Yaskawa INFORM job: R1_W49-52-A5(180,0)KM-OK.JBI

/JOB
//NAME R1_W49-52-A5(180,0)KM-OK
///FOLDERNAME KRIS-SCIANA
//POS
///NPOS 116,116,0,8,0,0
///TOOL 0
///POSTYPE PULSE
///PULSE
C00000=236346,-93771,-119067,-15606,106110,52447
C00001=224522,-84676,-111717,21504,108396,-36823
C00002=223323,-76354,-80310,30853,97883,-38151
C00003=223323,-76354,-80296,30852,97876,-38153
C00004=224728,-76958,-80577,30799,97249,-37774
C00005=223323,-76354,-80296,30852,97876,-38153
C00006=223323,-76341,-79339,30801,97373,-38291
C00007=223323,-76354,-80296,30852,97876,-38153
C00008=212037,-83911,-83077,30593,100081,-41994
C00009=212037,-83786,-81846,30518,99482,-42157
C00010=212037,-83911,-83077,30593,100081,-41994
C00011=241412,-119790,-112905,4528,90278,-34927
C00012=241412,-120659,-108380,4524,87055,-35044
C00013=241412,-118950,-107832,4524,87594,-35023
C00014=241412,-120659,-108380,4524,87055,-35044
C00015=241361,-125463,-113452,4527,87710,-35038
C00016=194879,-88434,-95721,7341,99248,-50176
C00017=197359,-87135,-94304,7246,98826,-49360
C00018=197775,-85843,-93756,7239,99114,-49203
C00019=197359,-87135,-94304,7246,98826,-49360
C00020=197359,-86577,-97024,7299,100771,-49245
C00021=203638,-64502,-86768,7203,105226,-46867
C00022=203638,-66884,-80001,7025,99877,-47180
C00023=203638,-66998,-79410,7014,99457,-47204
C00024=203638,-66468,-81766,7061,101167,-47106
C00025=189796,-64404,-88301,-2122,101648,-53086
C00026=192138,-63897,-80248,-2321,97017,-52239
C00027=192407,-63174,-79874,-2350,97166,-52152
C00028=192138,-63897,-80248,-2321,97017,-52239
C00029=192138,-62980,-82881,-2336,99107,-52278
C00030=196867,-49117,-75283,-2865,101696,-50791
C00031=196581,-52073,-70506,-2790,97234,-50782
C00032=196581,-52191,-70054,-2789,96895,-50774
C00033=196581,-52073,-70506,-2790,97234,-50782
C00034=196581,-46594,-80683,-2903,106301,-50992
C00035=236346,-93771,-119067,-15606,106110,52447
C00036=190859,-30717,-61907,-2252,102738,-52513
C00037=190859,-32261,-58668,-2226,99953,-52462
C00038=190859,-32540,-57932,-2222,99357,-52451
C00039=190859,-32848,-57040,-2218,98651,-52442
C00040=190859,-32743,-57355,-2220,98898,-52446
C00041=188695,-29142,-54935,-1991,99204,-53158
C00042=188695,-29402,-54164,-1988,98596,-53150
C00043=189471,-30718,-55056,-2070,98486,-52895
C00044=189092,-29546,-56142,-2024,99747,-53036
C00045=236346,-93771,-119067,-15606,106110,52447
C00046=196676,-46951,-80505,-2931,106009,-50708
C00047=226089,-87681,-87164,-16683,91869,41842
C00048=226089,-84980,-73215,-16676,84961,42778
C00049=222722,-83294,-69193,-16494,82730,41887
C00050=221384,-82519,-67534,-16419,81860,41530
C00051=221384,-82165,-66497,-16435,81422,41587
C00052=221384,-82519,-67534,-16419,81860,41530
C00053=220217,-82025,-67321,-16328,81744,41131
C00054=222131,-82891,-67940,-16470,82068,41767
C00055=218079,-90110,-72371,-12430,77203,39678
C00056=219704,-89894,-70139,-16382,79423,41260
C00057=219704,-89630,-69485,-16394,79165,41293
C00058=219704,-89894,-70139,-16382,79423,41260
C00059=218644,-89437,-69955,-16295,79329,40895
C00060=219704,-89894,-70139,-16382,79423,41260
C00061=221324,-92979,-76952,-12767,79023,40635
C00062=224587,-85889,-68614,-24649,81564,25677
C00063=224756,-83416,-64587,-24725,80512,25960
C00064=225339,-73949,-64106,-24638,87887,18307
C00065=226448,-82892,-63168,-24845,80468,26604
C00066=224819,-83008,-64496,-24719,80671,25950
C00067=225614,-76486,-63729,-24655,86567,18681
C00068=224629,-78708,-62826,-24669,84723,18698
C00069=225940,-68221,-57039,-24546,91074,32118
C00070=225024,-67480,-55852,-25246,95579,30588
C00071=225380,-76131,-59905,-25972,90581,27759
C00072=227101,-80482,-61144,-27753,88274,27425
C00073=225092,-75884,-57990,-29524,93980,25291
C00074=225490,-76153,-56481,-32832,88680,45115
C00075=225790,-75181,-58526,-32836,90285,44768
C00076=229050,-65408,-68692,-33536,101085,42880
C00077=230175,-63026,-84940,-35665,110860,40157
C00078=230138,-62898,-84918,-18541,99850,-36366
C00079=200601,-94229,-88213,1189,74472,-70745
C00080=200596,-94343,-86321,1199,73250,-70760
C00081=197671,-88605,-83096,1980,74270,-71770
C00082=195055,-82443,-79357,2670,75208,-72661
C00083=195099,-79673,-78401,2650,76040,-72625
C00084=204881,-52827,-65216,-6698,94281,-70293
C00085=196276,-62415,-68369,-628,83095,-72386
C00086=192341,-68440,-69414,3377,76385,-73570
C00087=192211,-66934,-68275,3411,76464,-73615
C00088=182841,-52271,-60438,13877,87086,-75412
C00089=190362,-40266,-53341,11309,86676,-73013
C00090=197861,-61500,-70436,1888,80400,-71610
C00091=209863,-89114,-92212,5168,89649,-66965
C00092=207997,-88203,-88549,6351,90131,-67524
C00093=201449,-78097,-83040,6985,92456,-69601
C00094=207997,-88240,-91061,6359,91649,-67447
C00095=228040,-108064,-102188,4192,87018,-60905
C00096=228112,-108053,-98628,4191,84835,-60953
C00097=219137,-101130,-95094,5195,86737,-63923
C00098=219137,-101703,-101195,5196,90183,-63781
C00099=214163,-101436,-96902,5723,88024,-65549
C00100=223035,-106938,-98576,4767,85658,-62646
C00101=223334,-107497,-100891,4730,86775,-62503
C00102=234921,-111060,-102133,3384,85128,-58640
C00103=235893,-110382,-100016,3269,84135,-58337
C00104=231608,-107829,-97339,12798,85544,-59388
C00105=223049,-95785,-95165,13566,91657,-61693
C00106=207574,-109422,-93472,27956,81376,-52899
C00107=219850,-54284,-73540,20701,118189,-64721
C00108=225869,-58194,-70692,20930,113190,-63323
C00109=219200,-94491,-85020,22840,89314,-46959
C00110=218101,-98890,-83982,26703,77531,-49761
C00111=221879,-76770,-74746,25704,81466,-47442
C00112=209721,-86136,-82329,27503,85211,-51165
C00113=230175,-51837,-95722,-39836,120784,36248
C00114=142430,-51837,-95722,-39836,120784,36248
C00115=142268,-143669,-120901,-39836,-2332,36248
BC00000=398177,21437,1035409
BC00001=398177,21437,1035409
BC00002=394644,68751,1035406
BC00003=394644,68751,1035406
BC00004=394644,68751,1035406
BC00005=394644,68751,1035406
BC00006=394644,68751,1035406
BC00007=394644,68751,1035406
BC00008=394644,68751,1035406
BC00009=394644,68751,1035406
BC00010=394644,68751,1035406
BC00011=394644,68751,1035406
BC00012=394644,68751,1035406
BC00013=394645,68750,1035403
BC00014=394644,68751,1035406
BC00015=394644,68751,1035406
BC00016=394644,68751,1035406
BC00017=394644,68751,1035406
BC00018=394644,68751,1035406
BC00019=394644,68751,1035406
BC00020=394644,68751,1035406
BC00021=394644,68751,1035406
BC00022=394644,68751,1035406
BC00023=394644,68751,1035406
BC00024=394644,68751,1035406
BC00025=394644,68751,1035406
BC00026=394644,68751,1035404
BC00027=394644,68751,1035404
BC00028=394644,68751,1035404
BC00029=394644,68751,1035404
BC00030=394644,68751,1035404
BC00031=394644,68751,1035404
BC00032=394644,68751,1035404
BC00033=394644,68751,1035404
BC00034=394644,68751,1035404
BC00035=398177,21437,1035409
BC00036=394654,68622,1035404
BC00037=394654,68622,1035404
BC00038=394654,68622,1035404
BC00039=394654,68622,1035404
BC00040=394654,68622,1035404
BC00041=394654,68622,1035404
BC00042=394654,68622,1035404
BC00043=394654,68622,1035404
BC00044=394653,68623,1035402
BC00045=398177,21437,1035409
BC00046=394654,68622,1035404
BC00047=398174,31874,1075175
BC00048=398174,31874,1075175
BC00049=398174,31874,1075175
BC00050=398174,31874,1075175
BC00051=398174,31874,1075175
BC00052=398174,31874,1075175
BC00053=398174,31874,1075175
BC00054=398174,31874,1075175
BC00055=398174,31874,1075175
BC00056=398174,31874,1075175
BC00057=398174,31874,1075175
BC00058=398174,31874,1075175
BC00059=398174,31874,1075175
BC00060=398174,31874,1075175
BC00061=398174,31874,1075175
BC00062=398174,45849,1075175
BC00063=398174,40485,1075175
BC00064=396736,36940,1075174
BC00065=398174,38340,1075175
BC00066=398174,38340,1075175
BC00067=396736,36940,1075174
BC00068=396736,36940,1075174
BC00069=396735,36938,1075175
BC00070=396735,36938,1075175
BC00071=396735,36938,1075175
BC00072=396735,36938,1075175
BC00073=396735,36938,1075175
BC00074=398174,45701,1075175
BC00075=398174,51572,1075175
BC00076=398174,51572,1075175
BC00077=398174,51572,1075175
BC00078=398171,51587,1075141
BC00079=398171,51587,1075141
BC00080=398171,51587,1075141
BC00081=398171,51587,1075141
BC00082=398171,51587,1075141
BC00083=398171,51587,1075141
BC00084=398171,51587,1075141
BC00085=398171,51587,1075141
BC00086=398171,51587,1075141
BC00087=398171,51587,1075141
BC00088=398171,51587,1075141
BC00089=398171,51587,1075141
BC00090=398171,51587,1075141
BC00091=398171,51587,1075141
BC00092=398171,51587,1075141
BC00093=398171,51587,1075141
BC00094=398171,51587,1075141
BC00095=398171,51587,1075141
BC00096=398171,51587,1075141
BC00097=398171,51587,1075141
BC00098=398171,51587,1075141
BC00099=398171,86239,1075141
BC00100=398171,86239,1075141
BC00101=398171,86239,1075141
BC00102=398171,86239,1075141
BC00103=398171,86239,1075141
BC00104=398171,86239,1075141
BC00105=398171,86239,1075141
BC00106=398171,86239,1075141
BC00107=398171,86239,1075141
BC00108=398171,86239,1075141
BC00109=398171,86239,1075138
BC00110=398171,86239,1075141
BC00111=398171,86239,1075141
BC00112=398171,86239,1075141
BC00113=398174,51572,1075175
BC00114=398174,51572,1075175
BC00115=398174,51572,1075175
///POSTYPE BASE
///RECTAN
///RCONF 0,0,0,0,1,0,0,0,0,0,0,0,0,0,0,0,0,0,0,0,0,0,0,0
P00006=2.006,1.622,-0.565,0.0000,0.0000,0.0000
///RCONF 0,0,0,0,0,0,0,0,0,0,0,0,0,0,0,0,0,0,0,0,0,0,0,0
P00023=-2.957,-4.083,2.762,0.0000,0.0000,0.0000
P00025=3.643,0.007,-2.585,0.0000,0.0000,0.0000
P00026=2.644,0.055,-2.583,0.0000,0.0000,0.0000
P00027=2.278,0.099,-4.210,0.0000,0.0000,0.0000
P00028=-1.778,-0.182,-2.050,0.0000,0.0000,0.0000
P00030=-0.014,-0.768,0.131,0.0000,0.0000,0.0000
P00050=-0.123,2.174,-1.314,0.0000,0.0000,0.0000
//INST
///DATE 2024/09/16 12:20
///ATTR SC,RW
///GROUP1 RB1,BS1
NOP
'r1_W49-52-A5(180,0)
'Path S1195
SFTOF
MOVJ C00000 BC00000 VJ=10.00
MOVJ C00001 BC00001 VJ=20.00
MOVJ C00002 BC00002 VJ=20.00
MOVL C00003 BC00003 V=83.3
REFP 3 C00004 BC00004
CALL JOB:SEARCH-R1
SET P025 P006
SFTON P025
MOVL C00005 BC00005 V=60.0
REFP 3 C00006 BC00006
CALL JOB:SEARCH-R1
SET P025 P006
SFTON P025
MOVL C00007 BC00007 V=60.0
SFTOF
MOVL C00008 BC00008 V=83.3
REFP 3 C00009 BC00009
CALL JOB:SEARCH-R1
SET P026 P006
SFTON P026
MOVL C00010 BC00010 V=83.3
MOVL C00011 BC00011 V=83.3
MOVL C00012 BC00012 V=83.3
REFP 3 C00013 BC00013
CALL JOB:SEARCH-R1
SET P026 P006
SFTON P026
MOVL C00014 BC00014 V=83.3
SFTOF
MOVL C00015 BC00015 V=83.3
MOVL C00016 BC00016 V=166.7
MOVL C00017 BC00017 V=83.3
REFP 3 C00018 BC00018
CALL JOB:SEARCH-R1
SET P027 P006
SFTON P027
MOVL C00019 BC00019 V=83.3
MOVL C00020 BC00020 V=83.3
MOVL C00021 BC00021 V=83.3
MOVL C00022 BC00022 V=83.3
REFP 3 C00023 BC00023
CALL JOB:SEARCH-R1
SET P027 P006
SFTON P027
MOVL C00024 BC00024 V=83.3
MOVL C00025 BC00025 V=166.7
SFTOF
MOVL C00026 BC00026 V=166.7
REFP 3 C00027 BC00027
CALL JOB:SEARCH-R1
SET P028 P006
SFTON P028
MOVL C00028 BC00028 V=83.3
MOVL C00029 BC00029 V=83.3
MOVL C00030 BC00030 V=83.3
MOVL C00031 BC00031 V=83.3
REFP 3 C00032 BC00032
CALL JOB:SEARCH-R1
SET P028 P006
SFTON P028
MOVL C00033 BC00033 V=83.3
MOVL C00034 BC00034 V=83.3
SFTOF
MOVJ C00035 BC00035 VJ=25.00
'BP 100624
MOVJ C00036 BC00036 VJ=25.00
MOVL C00037 BC00037 V=166.7
MOVL C00038 BC00038 V=60.0
REFP 3 C00039 BC00039
CALL JOB:SEARCH-R1
SET P050 P006
SFTON P050
MOVL C00040 BC00040 V=60.0
MOVL C00041 BC00041 V=166.7
MOVL C00042 BC00042 V=60.0
REFP 3 C00043 BC00043
CALL JOB:SEARCH-R1
SET P050 P006
SFTON P050
MOVL C00044 BC00044 V=60.0
SFTOF
MOVJ C00045 BC00045 VJ=25.00
'KONIEC BP 100624
MOVJ C00046 BC00046 VJ=25.00
MOVJ C00047 BC00047 VJ=25.00
MOVJ C00048 BC00048 VJ=10.00
MOVJ C00049 BC00049 VJ=10.00
MOVL C00050 BC00050 V=60.0
REFP 3 C00051 BC00051
CALL JOB:SEARCH-R1
SET P023 P006
SFTON P023
MOVL C00052 BC00052 V=60.0
REFP 3 C00053 BC00053
CALL JOB:SEARCH-R1
SET P023 P006
SFTON P023
MOVL C00054 BC00054 V=60.0
SFTOF
MOVL C00055 BC00055 V=100.0
MOVL C00056 BC00056 V=60.0
REFP 3 C00057 BC00057
CALL JOB:SEARCH-R1
SET P030 P006
SFTON P030
MOVL C00058 BC00058 V=60.0
REFP 3 C00059 BC00059
CALL JOB:SEARCH-R1
SET P030 P006
MOVL C00060 BC00060 V=60.0
MOVL C00061 BC00061 V=166.7
'Path W1196
SFTOF
SFTON P023
CALL JOB:COFNIJ_DRUT
MOVJ C00062 BC00062 VJ=10.00
MOVJ C00063 BC00063 VJ=10.00
MOVL C00064 BC00064 V=100.0 PL=0
REFP 1 C00065 BC00065
REFP 2 C00066 BC00066
MACRO1 MJ#(0) ARGF9
ARCON
MOVL C00067 BC00067 V=10.0
MOVL C00068 BC00068 V=10.0
MOVL C00069 BC00069 V=10.0
SFTON P030
MOVL C00070 BC00070 V=10.0
MOVL C00071 BC00071 V=10.0
MOVL C00072 BC00072 V=10.0
MOVL C00073 BC00073 V=10.0
ARCOF
MOVL C00074 BC00074 V=100.0
MOVL C00075 BC00075 V=166.7
SFTOF
MOVJ C00076 BC00076 VJ=10.00
MOVJ C00077 BC00077 VJ=10.00
'SPAWANIE SPION PRZERYWANYCH
MOVJ C00078 BC00078 VJ=20.00
MACRO1 MJ#(0) ARGF6
MOVJ C00079 BC00079 VJ=20.00
SFTON P028
MOVJ C00080 BC00080 VJ=20.00
ARCON
MOVL C00081 BC00081 V=16.7
MOVL C00082 BC00082 V=16.7
ARCOF
MOVL C00083 BC00083 V=50.0
MOVL C00084 BC00084 V=50.0
ARCON
MOVL C00085 BC00085 V=11.7
MOVL C00086 BC00086 V=11.7
MACRO1 MJ#(0) ARGF6
ARCON
MACRO1 MJ#(0) ARGF6
MOVL C00087 BC00087 V=11.7
SFTON P050
MOVL C00088 BC00088 V=11.7
ARCON
WVON WEV#(50)
MACRO1 MJ#(0) ARGF12
MOVL C00089 BC00089 V=13.3
ARCOF
WVOF
MOVL C00090 BC00090 V=83.3
MACRO1 MJ#(0) ARGF6
MOVJ C00091 BC00091 VJ=20.00
SFTOF
SFTON P027
MOVJ C00092 BC00092 VJ=20.00
ARCON
MOVL C00093 BC00093 V=13.3
ARCOF
MOVJ C00094 BC00094 VJ=20.00
MOVJ C00095 BC00095 VJ=20.00
MOVJ C00096 BC00096 VJ=20.00
ARCON
MOVL C00097 BC00097 V=13.3
ARCOF
MOVJ C00098 BC00098 VJ=20.00
SFTOF
SFTON P026
MOVJ C00099 BC00099 VJ=20.00
ARCON
MOVL C00100 BC00100 V=13.3
ARCOF
MOVJ C00101 BC00101 VJ=20.00
MOVJ C00102 BC00102 VJ=20.00
MOVJ C00103 BC00103 VJ=20.00
ARCON
MOVL C00104 BC00104 V=16.7
ARCOF
MOVJ C00105 BC00105 VJ=20.00
SFTOF
MOVJ C00106 BC00106 VJ=20.00
MACRO1 MJ#(0) ARGF7
MOVJ C00107 BC00107 VJ=25.00
SFTON P025
MOVJ C00108 BC00108 VJ=20.00
ARCON
MOVL C00109 BC00109 V=8.3
MOVL C00110 BC00110 V=8.3
MOVL C00111 BC00111 V=8.3
ARCOF
MOVJ C00112 BC00112 VJ=20.00
SFTOF
MOVJ C00113 BC00113 VJ=10.00
MOVJ C00114 BC00114 VJ=50.00
MOVJ C00115 BC00115 VJ=100.00
SFTOF
END
